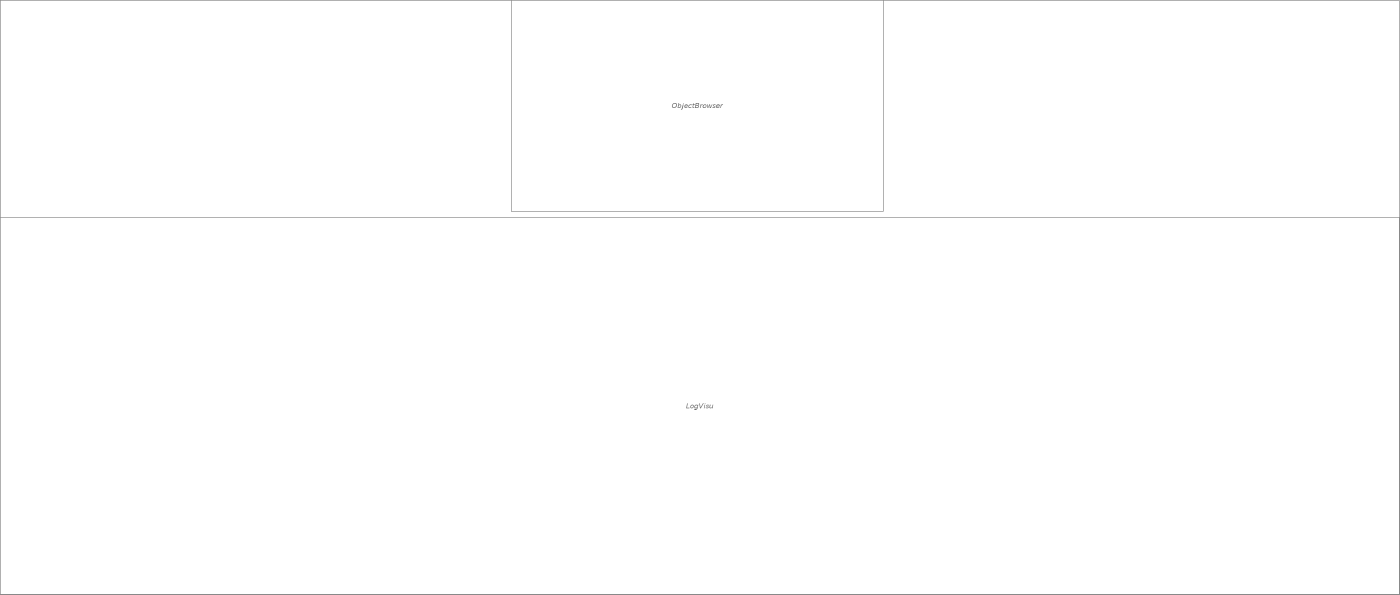
VISUALIZATION LandingPage  // 2000x850
    Frame (0,310 2000x540)
        shows LogVisu()
    Frame (730,0 532x302)
        shows ObjectBrowser()
END_VISUALIZATION

(* stored: Version 1.1.0.1, ProductVersion 3.1.4024.12
   Visu LandingPage: Id {06a96644-e797-418e-ba03-572ce05adbec} *)
